FUNCTION_BLOCK FB_WriteParameterNC_TestDouble IMPLEMENTS  I_WriteParameter
VAR
    bError : BOOL;
    nErrorID : UDINT := 26000;
END_VAR

{warning 'Add property implementation'}
PROPERTY Aborted : BOOL
GET
END_GET
END_PROPERTY

{warning 'Add property implementation'}
PROPERTY Active : BOOL
GET
END_GET
END_PROPERTY

{warning 'Add property implementation'}
PROPERTY Busy : BOOL
GET
END_GET
END_PROPERTY

{warning 'Add property implementation'}
PROPERTY Done : BOOL
GET
END_GET
END_PROPERTY

{warning 'Add property implementation'}
PROPERTY Error : BOOL
GET
Error := bError;
END_GET
SET
bError := Error;
END_SET
END_PROPERTY

{warning 'Add property implementation'}
PROPERTY ErrorID : UDINT
GET
ErrorId := nErrorID;
END_GET
SET
nErrorId := ErrorID;
END_SET
END_PROPERTY

{warning 'Add property implementation'}
PROPERTY Message : T_MAXSTRING
GET
END_GET
END_PROPERTY

{warning 'Add method implementation '}
METHOD WriteParameter
VAR_INPUT
    ParameterNumber	: MC_AxisParameter;
    ParameterValue	: LREAL;
END_VAR
END_METHOD

END_FUNCTION_BLOCK

(* stored: Version 1.1.0.1
   POU FB_WriteParameterNC_TestDouble: Id {585873b6-7f78-428d-a151-a1ef70c92da6}, SpecialFunc None
   Property Aborted: Id {a647de76-3753-480c-b146-053a5b27a657}
   Get Get: Id {f7abb830-9a25-4afb-9ea2-6000257057b8}
   Property Active: Id {90b6a55e-8e9a-42c4-8096-3c254f7ecb5e}
   Get Get: Id {33eaa287-f028-483e-8608-5d0fbbe09d1f}
   Property Busy: Id {4afd0ea4-3fd3-4807-acfe-15e5317d693a}
   Get Get: Id {9be62834-716a-4d14-b412-096e62ebc2aa}
   Property Done: Id {8cccf0fc-15e9-4486-ad58-bc1102c04d11}
   Get Get: Id {2316b095-17cd-41ef-bd20-2763e4afd9da}
   Property Error: Id {934a8d8d-b58c-44e1-830a-73770afa6528}
   Get Get: Id {58d2b9e0-14f3-4404-b4e8-100826546820}
   Set Set: Id {95037f81-3a6e-4c64-9295-a0d719594b5d}
   Property ErrorID: Id {ad4ca2dc-8103-4fda-a9ea-b3238abf15e8}
   Get Get: Id {2ef6794c-2dd4-4581-9c32-6d34f6e80aaf}
   Set Set: Id {bc55ff4a-ea9e-44be-8bc8-e11a9c0014c6}
   Property Message: Id {1f58cb4a-2627-48c6-be45-4d4613f93620}
   Get Get: Id {716e9cf0-1795-4fd3-a23a-4c4dc3a39f04}
   Method WriteParameter: Id {26b94086-a1ed-4735-b189-866b38035099} *)
